TYPE ST_Curtain_ip :
STRUCT
	OpenCmd AT%I* : BOOL;
	CloseCmd AT%I* : BOOL;	
END_STRUCT
END_TYPE

(* stored: Version 1.1.0.1, ProductVersion 3.1.4024.12
   DUT ST_Curtain_ip: Id {8a5a58b4-1b02-45ae-a6df-eaa493e3d5b4} *)
